// TIA Portal project "QPLC_LADDER" (V16)

(* hardware
DEVICE "S7-1200 station_1"  S7-1200 Station
   slot 0: "Rack_0"  S7-1200 Rack  Rack  V1.0
   slot 1: "PLC_1"  CPU 1214C DC/DC/DC  6ES7 214-1AG40-0XB0  V4.4
   slot 2: "DI 8/DQ 8x24VDC_1"  6ES7 223-1BH32-0XB0  V2.0
*)

// ===== PLC "PLC_1"  CPU 1214C DC/DC/DC =====

VAR_GLOBAL   // PLC tag table "Default tag table"
   "start" AT %I0.0 : Bool;   // Botão começar produção
   "stop" AT %I0.1 : Bool;   // Botão parar produção
   "reset" AT %I0.2 : Bool;   // Botão Reset produção
   "chave" AT %I0.3 : Bool;   // Seleção Modo Automático/Manual
   "Emergência (NO)" AT %I0.4 : Bool;   // Botão de emergencia NO
   "Sen_Peça_Inicial" AT %I0.5 : Bool;   // Sensor detetor de peça
   "Sensor Posição 3" AT %I0.6 : Bool;
   "Sensor Posição 2" AT %I0.7 : Bool;
   "Sen_Gripper_Embaixo" AT %I1.0 : Bool;   // Sensor do braço avançado
   "Sen_Gripper_Em_Cima" AT %I1.1 : Bool;   // Sensor do braço Recuado
   "Sen_Garra_Função" AT %I1.2 : Bool;   // Posição da garra
   "Sensor Posição 1" AT %I1.3 : Bool;   // Posição 1 do braço
   "Prato_Rec" AT %I1.4 : Bool;
   "Prato_Avanc" AT %I1.5 : Bool;
   "Btn_NC_Em" AT %I1.6 : Bool;   // Botão de emergencia NO
   "Pressostato" AT %I1.7 : Bool;
   "LedStart_KA1" AT %Q0.0 : Bool;
   "LedReset_KA2" AT %Q0.1 : Bool;
   "LedQ1_KA3" AT %Q0.2 : Bool;   // Também vai para a o sinalizador da torre
   "LEDQ2_KA4" AT %Q0.3 : Bool;
   "Braço_Direita" AT %Q0.4 : Bool;   // Ordem mover braço para esquerda
   "Braço_Esquerda" AT %Q0.5 : Bool;   // Ordem mover braço para direita
   "Braço_Ação" AT %Q0.6 : Bool;   // Ordem de avanço do braço
   "Garra_AbertaKA8" AT %Q0.7 : Bool;   // Ordem abertura da garra
   "Prato_Rec_KA9" AT %Q1.0 : Bool;   // Ordem recuar o prato
   "Prato_Avan_KA10" AT %Q1.1 : Bool;   // Ordem avançar o prato
   "Valv_KA11" AT %Q1.2 : Bool;
   "System_Byte" AT %MB1 : Byte;
   "FirstScan" AT %M1.0 : Bool;
   "DiagStatusUpdate" AT %M1.1 : Bool;
   "AlwaysTRUE" AT %M1.2 : Bool;
   "AlwaysFALSE" AT %M1.3 : Bool;
   "E_1" AT %M2.0 : Bool;
   "E_2" AT %M2.1 : Bool;
   "E_3" AT %M2.2 : Bool;
   "E_4" AT %M2.3 : Bool;
   "E_5" AT %M2.4 : Bool;
   "E_6" AT %M2.5 : Bool;
   "E_7" AT %M2.6 : Bool;
   "E_8" AT %M2.7 : Bool;
   "E_9" AT %M3.0 : Bool;
   "E_10" AT %M3.1 : Bool;
   "E_11" AT %M3.2 : Bool;
END_VAR

// folder: System blocks/Program resources

DATA_BLOCK "Cooldown para Direita"   // DB1
{ S7_Optimized_Access := 'TRUE' }
AUTHOR : Simatic
FAMILY : IEC
NAME : IEC_TMR
VERSION : 1.0
// stored: InstanceOfName IEC_TIMER
"IEC_TIMER"
BEGIN
END_DATA_BLOCK

DATA_BLOCK "Bit_ON_E2"   // DB2
{ S7_Optimized_Access := 'TRUE' }
AUTHOR : Simatic
FAMILY : IEC
NAME : IEC_TMR
VERSION : 1.0
// stored: InstanceOfName IEC_TIMER
"IEC_TIMER"
BEGIN
END_DATA_BLOCK

DATA_BLOCK "Cooldown_Para_Voltar"   // DB3
{ S7_Optimized_Access := 'TRUE' }
AUTHOR : Simatic
FAMILY : IEC
NAME : IEC_TMR
VERSION : 1.0
// stored: InstanceOfName IEC_TIMER
"IEC_TIMER"
BEGIN
END_DATA_BLOCK

DATA_BLOCK "Tempo para Descer Peça"   // DB4
{ S7_Optimized_Access := 'TRUE' }
AUTHOR : Simatic
FAMILY : IEC
NAME : IEC_TMR
VERSION : 1.0
// stored: InstanceOfName IEC_TIMER
"IEC_TIMER"
BEGIN
END_DATA_BLOCK

DATA_BLOCK "Cooldown_E7"   // DB5
{ S7_Optimized_Access := 'TRUE' }
AUTHOR : Simatic
FAMILY : IEC
NAME : IEC_TMR
VERSION : 1.0
// stored: InstanceOfName IEC_TIMER
"IEC_TIMER"
BEGIN
END_DATA_BLOCK

DATA_BLOCK "2s"   // DB6
{ S7_Optimized_Access := 'TRUE' }
AUTHOR : Simatic
FAMILY : IEC
NAME : IEC_TMR
VERSION : 1.0
// stored: InstanceOfName IEC_TIMER
"IEC_TIMER"
BEGIN
END_DATA_BLOCK

DATA_BLOCK "Tempo para Soltar a Peça"   // DB7
{ S7_Optimized_Access := 'TRUE' }
AUTHOR : Simatic
FAMILY : IEC
NAME : IEC_TMR
VERSION : 1.0
// stored: InstanceOfName IEC_TIMER
"IEC_TIMER"
BEGIN
END_DATA_BLOCK

DATA_BLOCK "Tempo para Subir com Peça"   // DB8
{ S7_Optimized_Access := 'TRUE' }
AUTHOR : Simatic
FAMILY : IEC
NAME : IEC_TMR
VERSION : 1.0
// stored: InstanceOfName IEC_TIMER
"IEC_TIMER"
BEGIN
END_DATA_BLOCK

// folder: (top level)

FUNCTION "Geral - Peça 1" : Void   // FC1, LAD
{ S7_Optimized_Access := 'TRUE' }
VERSION : 0.1
BEGIN

REGION Network 1: Ordem Subir Braço
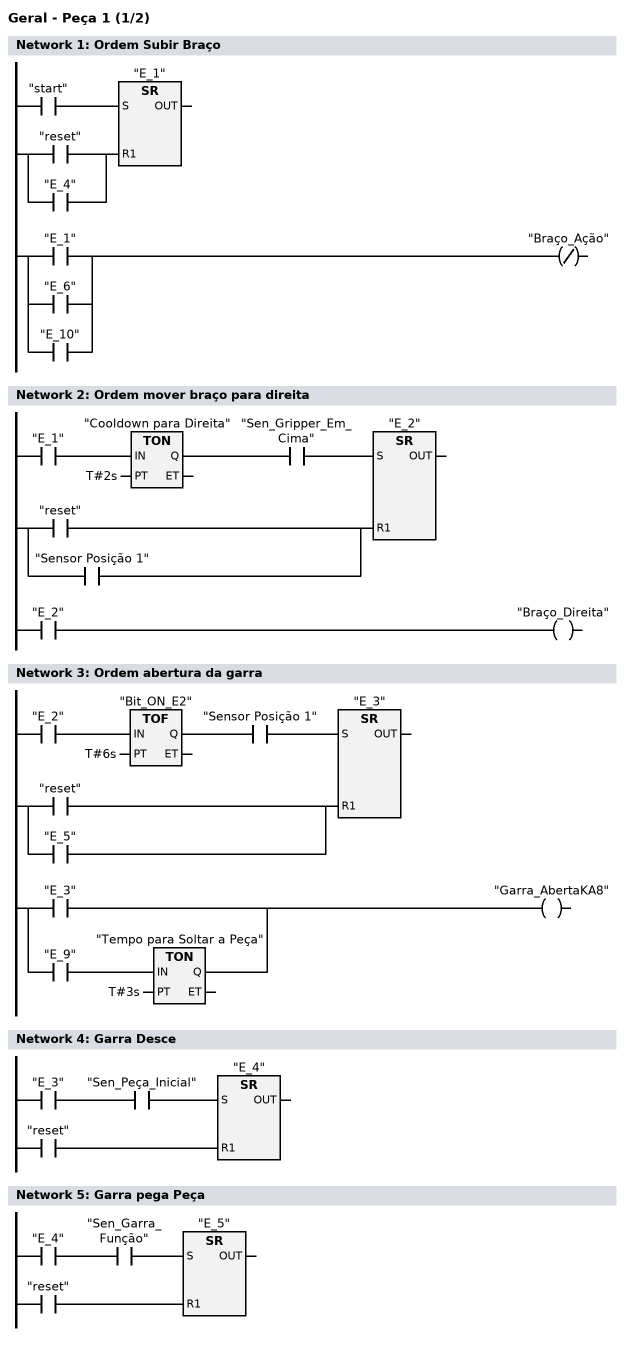
   RUNG wire#powerrail
      Contact( "start" )
      S_SR(operand := "E_1", r1 := wire#w1)
   END_RUNG
   RUNG wire#powerrail
      Contact( "reset" )
   END_RUNG wire#w1
   RUNG wire#powerrail
      Contact( "E_4" )
   END_RUNG wire#w1
   RUNG wire#powerrail
      Contact( "E_1" )
      wire#w2
      I_Coil( "Braço_Ação" )
   END_RUNG
   RUNG wire#powerrail
      Contact( "E_6" )
   END_RUNG wire#w2
   RUNG wire#powerrail
      Contact( "E_10" )
   END_RUNG wire#w2
   // the same network as SCL:
   IF "start" THEN
       "E_1" := TRUE;   // SR flip-flop
   END_IF;
   IF "reset" OR "E_4" THEN "E_1" := FALSE; END_IF;
   "Braço_Ação" := NOT ("E_1" OR "E_6" OR "E_10");
END_REGION

REGION Network 2: Ordem mover braço para direita
   "Cooldown para Direita".TON(IN := "E_1", PT := T#2s);
   IF "Cooldown para Direita".Q AND "Sen_Gripper_Em_Cima" THEN
       "E_2" := TRUE;   // SR flip-flop
   END_IF;
   IF "reset" OR "Sensor Posição 1" THEN "E_2" := FALSE; END_IF;
   "Braço_Direita" := "E_2";
END_REGION

REGION Network 3: Ordem abertura da garra
   "Bit_ON_E2".TOF(IN := "E_2", PT := T#6s);
   IF "Bit_ON_E2".Q AND "Sensor Posição 1" THEN
       "E_3" := TRUE;   // SR flip-flop
   END_IF;
   IF "reset" OR "E_5" THEN "E_3" := FALSE; END_IF;
   "Tempo para Soltar a Peça".TON(IN := "E_9", PT := T#3s);
   "Garra_AbertaKA8" := "E_3" OR "Tempo para Soltar a Peça".Q;
END_REGION

REGION Network 4: Garra Desce
   RUNG wire#powerrail
      Contact( "E_3" )
      Contact( "Sen_Peça_Inicial" )
      S_SR(operand := "E_4", r1 := wire#w1)
   END_RUNG
   RUNG wire#powerrail
      Contact( "reset" )
   END_RUNG wire#w1
   // the same network as SCL:
   IF "E_3" AND "Sen_Peça_Inicial" THEN
       "E_4" := TRUE;   // SR flip-flop
   END_IF;
   IF "reset" THEN "E_4" := FALSE; END_IF;
END_REGION

REGION Network 5: Garra pega Peça
   RUNG wire#powerrail
      Contact( "E_4" )
      Contact( "Sen_Garra_Função" )
      S_SR(operand := "E_5", r1 := wire#w1)
   END_RUNG
   RUNG wire#powerrail
      Contact( "reset" )
   END_RUNG wire#w1
   // the same network as SCL:
   IF "E_4" AND "Sen_Garra_Função" THEN
       "E_5" := TRUE;   // SR flip-flop
   END_IF;
   IF "reset" THEN "E_5" := FALSE; END_IF;
END_REGION

REGION Network 6: Garra sobe com peça
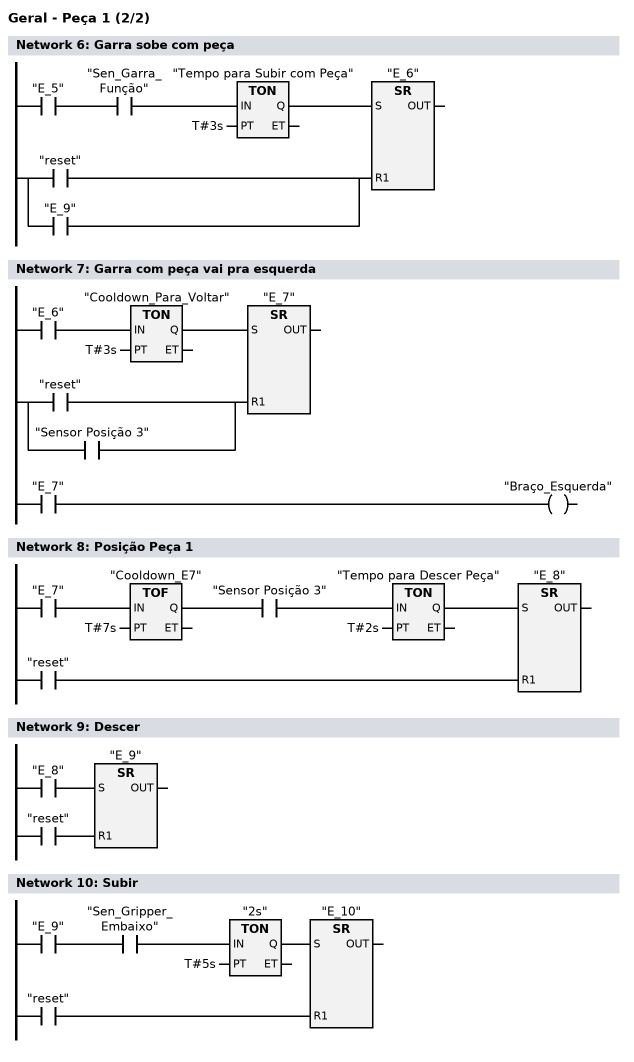
   "Tempo para Subir com Peça".TON(IN := "E_5" AND "Sen_Garra_Função", PT := T#3s);
   IF "Tempo para Subir com Peça".Q THEN
       "E_6" := TRUE;   // SR flip-flop
   END_IF;
   IF "reset" OR "E_9" THEN "E_6" := FALSE; END_IF;
END_REGION

REGION Network 7: Garra com peça vai pra esquerda
   "Cooldown_Para_Voltar".TON(IN := "E_6", PT := T#3s);
   IF "Cooldown_Para_Voltar".Q THEN
       "E_7" := TRUE;   // SR flip-flop
   END_IF;
   IF "reset" OR "Sensor Posição 3" THEN "E_7" := FALSE; END_IF;
   "Braço_Esquerda" := "E_7";
END_REGION

REGION Network 8: Posição Peça 1
   "Cooldown_E7".TOF(IN := "E_7", PT := T#7s);
   "Tempo para Descer Peça".TON(IN := "Cooldown_E7".Q AND "Sensor Posição 3", PT := T#2s);
   IF "Tempo para Descer Peça".Q THEN
       "E_8" := TRUE;   // SR flip-flop
   END_IF;
   IF "reset" THEN "E_8" := FALSE; END_IF;
END_REGION

REGION Network 9: Descer
   RUNG wire#powerrail
      Contact( "E_8" )
      S_SR(operand := "E_9", r1 := wire#w1)
   END_RUNG
   RUNG wire#powerrail
      Contact( "reset" )
   END_RUNG wire#w1
   // the same network as SCL:
   IF "E_8" THEN
       "E_9" := TRUE;   // SR flip-flop
   END_IF;
   IF "reset" THEN "E_9" := FALSE; END_IF;
END_REGION

REGION Network 10: Subir
   "2s".TON(IN := "E_9" AND "Sen_Gripper_Embaixo", PT := T#5s);
   IF "2s".Q THEN
       "E_10" := TRUE;   // SR flip-flop
   END_IF;
   IF "reset" THEN "E_10" := FALSE; END_IF;
END_REGION
END_FUNCTION

FUNCTION "Outputs" : Void   // FC2, LAD
{ S7_Optimized_Access := 'TRUE' }
VERSION : 0.1
BEGIN
END_FUNCTION

FUNCTION "Timers" : Void   // FC3, LAD
{ S7_Optimized_Access := 'TRUE' }
VERSION : 0.1
BEGIN
END_FUNCTION

ORGANIZATION_BLOCK "Main"   // OB1, LAD, ProgramCycle
TITLE = "Main Program Sweep (Cycle)"
{ S7_Optimized_Access := 'TRUE' }
VERSION : 0.1
// EXTRUTURA DO PROGRAMA
   VAR_INPUT
      Initial_Call : Bool;   // Initial call of this OB
      Remanence : Bool;   // =True, if remanent data are available
   END_VAR
BEGIN

REGION Network 1
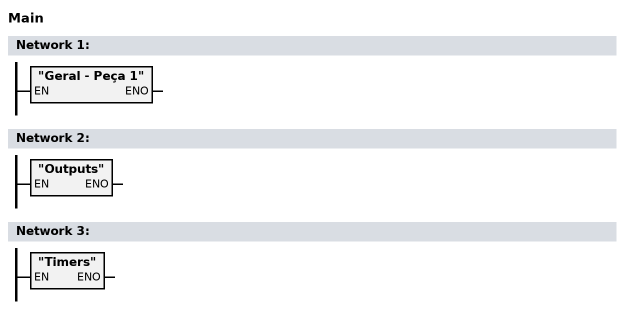
   RUNG wire#powerrail
      "Geral - Peça 1"()
   END_RUNG
   // the same network as SCL:
   "Geral - Peça 1"();
END_REGION

REGION Network 2
   RUNG wire#powerrail
      "Outputs"()
   END_RUNG
   // the same network as SCL:
   "Outputs"();
END_REGION

REGION Network 3
   RUNG wire#powerrail
      "Timers"()
   END_RUNG
   // the same network as SCL:
   "Timers"();
END_REGION
END_ORGANIZATION_BLOCK